TYPE ST_GCSingleProcessStageTimeConfig :
STRUCT
	TargetTime : TIME;
	Timeout : TIME;
END_STRUCT
END_TYPE

(* stored: Version 1.1.0.1, ProductVersion 3.1.4026.18
   DUT ST_GCSingleProcessStageTimeConfig: Id {f84ff372-3046-4d7d-aeef-defe2126d07e} *)
